PROGRAM P_DecDruck
VAR
END_VAR

IF DB6.rDrahthalterSchliessdruck > 0.9 THEN
	DB6.rDrahthalterSchliessdruck := DB6.rDrahthalterSchliessdruck - 0.5;
END_IF

END_PROGRAM

(* stored: Version 1.1.0.1, ProductVersion 3.1.4024.3
   POU P_DecDruck: Id {c3bd9a66-aed8-4c93-9650-a12876778b96}, SpecialFunc None *)
